PROGRAM MASTER_CTR
VAR
	//check status from finish state
	UR3FinishState : BOOL:= FALSE;
	UR5FinishState : BOOL:= FALSE;
	finish_state : BOOL:=FALSE;
	//var state to norm mode
	STATE :INT:=-1;
	//instance of sub state machines
	UR3_StateMachine :UR3_StateMachine;
	UR5_StateMachine :UR5_StateMachine;
	Vision_StateMachine : Vision_StateMachine;
	
	//instance of Qrob
	//QRob_StateMachine : QRob_StateMachine;
END_VAR

VAR_INPUT
	//vars to control the main stata machine
	  user_select_state : INT:=-1;
	  user_init: BOOL:=FALSE;
      User_Test_Sate :INT:=-1;
	  EMERGENCY_STOP :BOOL:=FALSE;
	  
END_VAR

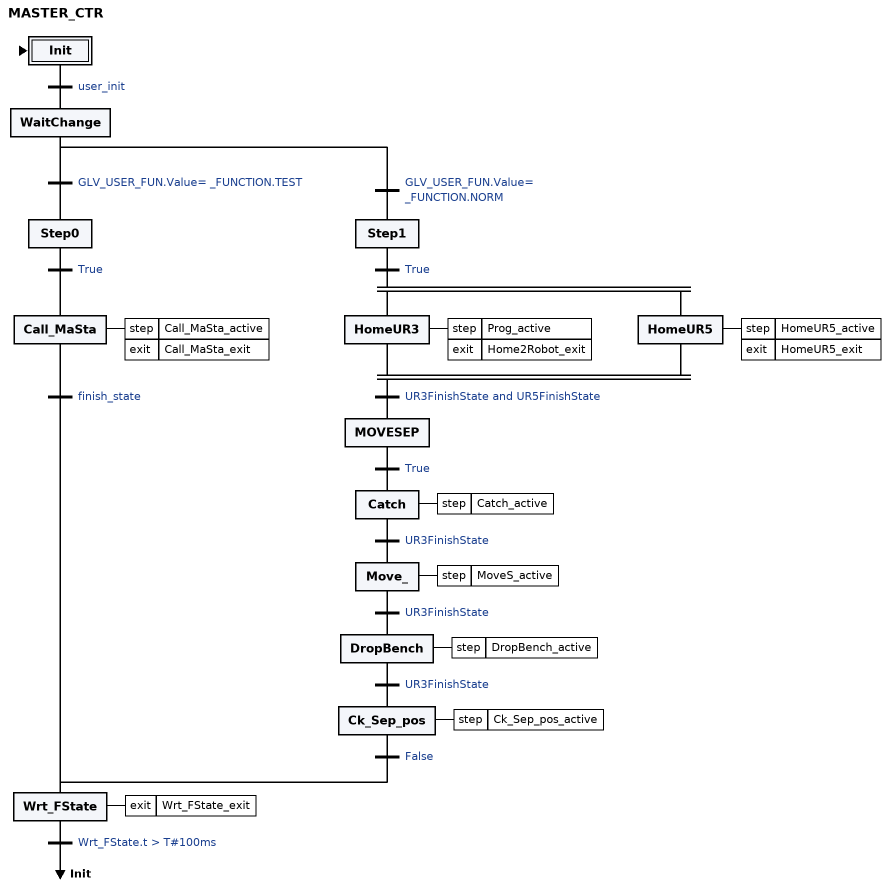
INITIAL_STEP Init:
END_STEP
TRANSITION FROM Init TO WaitChange
    := user_init;
END_TRANSITION
STEP WaitChange:
END_STEP
TRANSITION FROM WaitChange TO Step0
    := GLV_USER_FUN.Value= _FUNCTION.TEST;
END_TRANSITION
// macro TestMode begins
STEP Step0:
END_STEP
TRANSITION FROM Step0 TO Call_MaSta
    := True;
END_TRANSITION
STEP Call_MaSta:
    Call_MaSta_active(N);  // step action
    Call_MaSta_exit(P0);  // exit action
END_STEP
TRANSITION FROM Call_MaSta TO Wrt_FState
    := finish_state;
END_TRANSITION
TRANSITION FROM WaitChange TO Step1
    := GLV_USER_FUN.Value= _FUNCTION.NORM;
END_TRANSITION
// macro NormMode begins
STEP Step1:
END_STEP
TRANSITION FROM Step1 TO (HomeUR3, HomeUR5)
    := True;
END_TRANSITION
STEP HomeUR3:
    Prog_active(N);  // step action
    Home2Robot_exit(P0);  // exit action
END_STEP
STEP HomeUR5:
    HomeUR5_active(N);  // step action
    HomeUR5_exit(P0);  // exit action
END_STEP
TRANSITION FROM (HomeUR3, HomeUR5) TO MOVESEP
    := UR3FinishState and UR5FinishState;
END_TRANSITION
// macro MovSeparator begins
STEP MOVESEP:
END_STEP
TRANSITION FROM MOVESEP TO Catch
    := True;
END_TRANSITION
STEP Catch:
    Catch_active(N);  // step action
END_STEP
TRANSITION FROM Catch TO Move_
    := UR3FinishState;
END_TRANSITION
STEP Move_:
    MoveS_active(N);  // step action
END_STEP
TRANSITION FROM Move_ TO DropBench
    := UR3FinishState;
END_TRANSITION
STEP DropBench:
    DropBench_active(N);  // step action
END_STEP
TRANSITION FROM DropBench TO Ck_Sep_pos
    := UR3FinishState;
END_TRANSITION
STEP Ck_Sep_pos:
    Ck_Sep_pos_active(N);  // step action
END_STEP
TRANSITION FROM Ck_Sep_pos TO Wrt_FState
    := False;
END_TRANSITION
STEP Wrt_FState:
    Wrt_FState_exit(P0);  // exit action
END_STEP
TRANSITION FROM Wrt_FState TO Init
    := Wrt_FState.t > T#100ms;
END_TRANSITION

ACTION Call_MaSta_active:
//cal UR3 state Machine
//UR3(init, state_to_exec,out_proces,out_global_state, out_internal_state
//IF User_Test_Sate <30 THEN
IF User_Test_Sate >0 and User_Test_Sate <30 THEN
Vision_StateMachine(init_:=TRUE, G_STATE:=User_Test_Sate, State_complete=>finish_state,Act_Gl_State=>VisionRetVarState.Actual_GLV_State,Act_In_State=>VisionRetVarState.Actual_In_State);
//Vision_StateMachine(init_:=TRUE, G_STATE:=User_Test_Sate);
//finish_state:=Vision_StateMachine.State_complete;
//VisionRetVarState.Actual_GLV_State:=Vision_StateMachine.Act_Gl_State;
//VisionRetVarState.Actual_In_State:=Vision_StateMachine.Act_In_State;
ELSIF User_Test_Sate >=30 AND User_Test_Sate<50 THEN
UR3_StateMachine(init_:=TRUE, G_STATE:=User_Test_Sate, State_complete=>finish_state,Act_Gl_State=>UR3RetVarState.Actual_GLV_State,Act_In_State=>UR3RetVarState.Actual_In_State);	
//UR3_StateMachine(init_:=TRUE, G_STATE:=User_Test_Sate);
//finish_state:= UR3_StateMachine.State_complete;
//UR3RetVarState.Actual_GLV_State:=UR3_StateMachine.Act_Gl_State;
//UR3RetVarState.Actual_In_State:=UR3_StateMachine.Act_In_State;
ELSIF User_Test_Sate >=50 AND User_Test_Sate < 100THEN	
UR5_StateMachine(init_:=TRUE, G_STATE:=User_Test_Sate, Num_Ctr_Cam:=-1,State_complete=>finish_state, Act_Gl_State=>UR5RetVarState.Actual_GLV_State,Act_In_State=>UR5RetVarState.Actual_In_State);	
//UR5_StateMachine(init_:=TRUE, G_STATE:=User_Test_Sate);
//finish_state:= UR5_StateMachine.State_complete;
//UR5RetVarState.Actual_GLV_State:=UR5_StateMachine.Act_Gl_State;
//UR5RetVarState.Actual_In_State:=UR5_StateMachine.Act_In_State;

ELSIF User_Test_Sate >=50 AND User_Test_Sate < 100THEN	
	//QRob_StateMachine(init_:=TRUE);
END_IF


//UR3_StateMachine(TRUE,User_Test_Sate);
END_ACTION

ACTION Call_MaSta_exit:
//reset satte variable
User_Test_Sate:=-1;
finish_state := False;
END_ACTION

ACTION Catch_active:
//call respective state to ur3 robot
UR3_StateMachine(init_:=TRUE, G_STATE:=RCts.UR3CatchSeparator, State_complete=>UR3FinishState, Act_Gl_State=>UR3RetVarState.Actual_GLV_State,Act_In_State=>UR3RetVarState.Actual_In_State);
END_ACTION

ACTION Catch_exit:

END_ACTION

ACTION CatchSep_active:

END_ACTION

ACTION Ck_Sep_pos_active:
//call respective state to machine system
Vision_StateMachine(init_:=TRUE, G_STATE:=User_Test_Sate, State_complete=>finish_state,Act_Gl_State=>VisionRetVarState.Actual_GLV_State,Act_In_State=>VisionRetVarState.Actual_In_State);
END_ACTION

ACTION DropBench_active:
//call respective state to ur3 robot
UR3_StateMachine(init_:=TRUE, G_STATE:=RCts.UR3DropBench, State_complete=>UR3FinishState, Act_Gl_State=>UR3RetVarState.Actual_GLV_State,Act_In_State=>UR3RetVarState.Actual_In_State);
END_ACTION

ACTION Home2Robot_exit:
//reset the global state into instance state machine
UR3_StateMachine(init_:=FALSE, G_STATE:=RCts.RESET_STATE, State_complete=>UR3FinishState, Act_Gl_State=>UR3RetVarState.Actual_GLV_State,Act_In_State=>UR3RetVarState.Actual_In_State);
END_ACTION

ACTION HomeUR5_active:
//call respective state to ur5 robot
UR5_StateMachine(init_:=TRUE, G_STATE:=RCts.UR5Home, Num_Ctr_Cam:=-1,State_complete=>UR5FinishState, Act_Gl_State=>UR5RetVarState.Actual_GLV_State,Act_In_State=>UR5RetVarState.Actual_In_State);
END_ACTION

ACTION HomeUR5_exit:
//reset the global state into instance state machine
UR5_StateMachine(init_:=FALSE, G_STATE:=RCts.RESET_STATE, State_complete=>UR5FinishState, Act_Gl_State=>UR5RetVarState.Actual_GLV_State,Act_In_State=>UR5RetVarState.Actual_In_State);
END_ACTION

ACTION MoveS_active:
//call respective state to ur3 robot
UR3_StateMachine(init_:=TRUE, G_STATE:=RCts.UR3Move, State_complete=>UR3FinishState, Act_Gl_State=>UR3RetVarState.Actual_GLV_State,Act_In_State=>UR3RetVarState.Actual_In_State);
END_ACTION

ACTION MOVESEP_exit:
//changet the state to exec
STATE := RCts.UR3CatchSeparator;
END_ACTION

ACTION Prog_active:
//call respective state to ur3 robot
UR3_StateMachine(init_:=TRUE, G_STATE:=RCts.UR3Home, State_complete=>UR3FinishState, Act_Gl_State=>UR3RetVarState.Actual_GLV_State,Act_In_State=>UR3RetVarState.Actual_In_State);
END_ACTION

ACTION Wrt_FState_exit:
//reset the main var to init all process
//user_init:= FALSE;
END_ACTION

END_PROGRAM

(* stored: Version 1.1.0.1, ProductVersion 3.1.4024.4
   POU MASTER_CTR: Id {39b1979e-a165-4845-9ea3-97e5376ed519}, SpecialFunc None
   Action Call_MaSta_active: Id {02ffcfc6-3e93-4e18-9827-f2c35ee01d92}
   Action Call_MaSta_exit: Id {271ab7ba-cf61-46f6-b987-8e435f4619a9}
   Action Catch_active: Id {10b672cc-7c6e-4fd0-ad71-256cf62a1524}
   Action Catch_exit: Id {f9030493-ffc3-4094-b92e-11122f2ae1e9}
   Action CatchSep_active: Id {3e93b9c6-7c9a-4241-8d83-f82e551b992a}
   Action Ck_Sep_pos_active: Id {2be05195-fe1e-4182-894b-a1c12f7d15a7}
   Action DropBench_active: Id {06657ecd-2b56-47ec-b5ab-6c22c5fb61b3}
   Action Home2Robot_exit: Id {ff592298-6852-48b6-b1bd-0c1841237dbe}
   Action HomeUR5_active: Id {ac8a5ef3-1ef2-468b-a2cf-4c4b6b64b5e6}
   Action HomeUR5_exit: Id {03e10426-8f90-440a-9f4e-82654e36d729}
   Action MoveS_active: Id {b75d9cc2-2934-4189-a49a-16e64e3be012}
   Action MOVESEP_exit: Id {e5175d0e-cfca-436d-a2c5-6737c3f81b7b}
   Action Prog_active: Id {f18f4223-866c-41ea-9aff-f8bce9bd7968}
   Action Wrt_FState_exit: Id {840b7518-2748-496f-bf4c-3516d5943755} *)
